FUNCTION_BLOCK SUB_DT_TIME (* IEC 61131-3 DATE_AND_TIME-TIME *)
  (* Standard: 61131-3 *)
  (* Version 0.0, 2004-12-15, JHC, Rockwell Automation, Converted from SRC format. *)
  (* Compiler header: package fb.rt.plc.math; *)
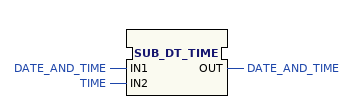
  VAR_INPUT
    IN1 : DATE_AND_TIME; (* Minuend *)
    IN2 : TIME; (* Subtrahend *)
  END_VAR
  VAR_OUTPUT
    OUT : DATE_AND_TIME; (* Difference *)
  END_VAR
END_FUNCTION_BLOCK
